{attribute 'qualified_only'}
{attribute 'strict'}
{attribute 'to_string'}
TYPE eLiftPins :
(
	In := 0,
	Out := 1,
	Unknown := 2
);
END_TYPE

(* stored: Version 1.1.0.1
   DUT eLiftPins: Id {9bd37c59-3295-496a-83fd-1779dfdf7c98} *)
